(* Schneider Machine Expert - Basic project 5 Run-2 Stop (1T) - Copy, file version 2.7.0.0 *)
(* ProjectInformations: Name=New project *)

HARDWARE
  Cpu 0: TM200C32R
  EthernetConfiguration: NetworkName=M200, IpAllocationMode=FixedAddress, IpAddress=0.0.0.0, SubnetMask=0.0.0.0
  SerialLineConfiguration: Baud=Baud19200, Parity=ParityEven, DataBits=DataBits8, StopBits=StopBits1, PhysicalMedium=PhysicalMediumRs485, TransmissionMode=TransmissionModeModbusRtu, SlaveId=1, Addressing=SlaveAddressing
  MastTask: UsePeriodScanMode=false, PeriodScan=100
  FastTask: Period=255
  CpuBehavior: StartingMode=StartAsPreviousState, AutoSaveRamOnEeprom=true, WatchdogPeriod=250

SYMBOLS  (address, symbol, comment, settings)
  %M0         "X"
  %M1         "T1 DN"
  %M2         "REST 2S"
  %M3         "C2 DN"
  %TM0        [Preset=7, Base=OneSecond]
  %I0.0       "START"
  %I0.1       "STOP"
  %Q0.0       "Motor"

POU New POU
  (* SectionNumber=1 *)

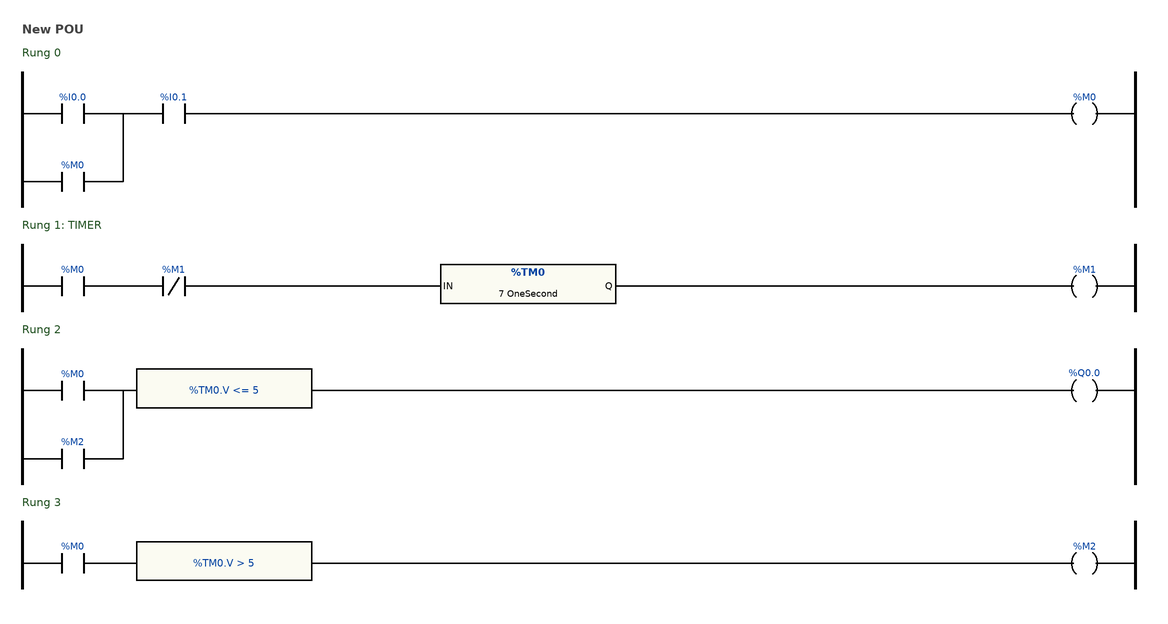

// Rung 0
  LD %I0.0
  OR %M0
  AND %I0.1
  ST %M0
  // as ST:
  //   %M0 := (%I0.0 OR %M0) AND %I0.1;

// Rung 1: TIMER
  BLK %TM0
  LD %M0
  ANDN %M1
  IN
  OUT_BLK
  LD Q
  ST %M1
  END_BLK
  // as ST:
  //   %TM0(IN := %M0 AND NOT %M1);
  //   %M1 := %TM0.Q;

// Rung 2
  LD %M0
  OR %M2
  AND [ %TM0.V <= 5 ]
  ST %Q0.0
  // as ST:
  //   %Q0.0 := (%M0 OR %M2) AND %TM0.V <= 5;

// Rung 3
  LD %M0
  AND [ %TM0.V > 5 ]
  ST %M2
  // as ST:
  //   %M2 := %M0 AND %TM0.V > 5;
